PROGRAM MAIN
VAR
	enclaveStart: BOOL;
	timerColumna: TON;
	posicionEst : ARRAY[1..2] OF REAL;
	distBaldas : distanciaBaldas();
END_VAR

(*
clumnas 1.6 - 1
filas 0.5-2.1
*)


IF GVLvar.botonStart THEN
	enclaveStart := TRUE;
	GVLvar.cinta := TRUE;
	distBaldas();
END_IF


IF enclaveStart THEN
	
	//si hay una caja en la enrada apr almacenar se prepara la grua
	IF GVLvar.sensorEntradaGrua THEN
		GVLvar.cinta := FALSE;
		posicionEst := posicionEstanteria();
		GVLvar.setPointX := posicionEst[1];
		GVLvar.setPointZ := posicionEst[2];
		//flanco de bajada en la senal de movimiento
		// xq si no se para automaticamente la grua al apsar al else
	ELSE
		GVLvar.setPointX := 0.0;
		GVLvar.setPointZ := 0.0;
	END_IF
	
	
END_IF

END_PROGRAM

(* stored: Version 1.1.0.1, ProductVersion 3.1.4024.15
   POU MAIN: Id {33819508-742b-4c1e-88e6-5bd373dd68ab}, SpecialFunc None *)
